{attribute addProperty BoxType "KL1352"}
{attribute addProperty Id "InputAT %I*BOOL000ErrorAT %I*BOOL000"}
{attribute addProperty CRC "1032597169"}
{attribute addProperty SizeInBites "0"}
{attribute addProperty SizeInBytes "0"}
TYPE Channel_3D8C2EB1 :
STRUCT
	{attribute addProperty Name "Input"}
	Input AT %I* : BOOL;
	{attribute addProperty Name "Error"}
	Error AT %I* : BOOL;
END_STRUCT
END_TYPE

(* stored: Version 1.2.0.0, ProductVersion 3.1.4024.9
   DUT Channel_3D8C2EB1: Id {a98f3940-7915-4d18-a041-123195008a24} *)
